// TIA Portal V20 export
TYPE "UDT_Tracability_Data"
   STRUCT
      Nb_of_Records { ExternalAccessible := 'False'; ExternalVisible := 'False'; ExternalWritable := 'False'} : Int := 100;
      Nb_of_Holes { ExternalAccessible := 'False'; ExternalVisible := 'False'; ExternalWritable := 'False'} : Int := 100;
      STRUCT_PART { ExternalAccessible := 'False'; ExternalVisible := 'False'; ExternalWritable := 'False'} : Array[0..99] of Struct
         Part_id : Int;
         Status : Int;
         Fail_code : Int;
         Raw_type : Int;
         Workpiece_holder_type : Int;
         Workpiece_holder_Nbr : Int;
         Datamatrix_code : Array[0..19] of Byte;
         Order_nbr : String[64];
         Ident_nbr : String[64];
         Batch_nbr : String[64];
         Operator_nbr : String[64];
         Comment : String[192];
         WOZ : Real;
         WOC : Real;
         Total_cycle_time : Int;
         Laser_cycle_time : Int;
         Measure_load_cycle_time : Int;
         STRUCT_HOLE : Array[0..99] of "UDT_Holes";
      END_STRUCT;
   END_STRUCT;
   // STRUCT_PART[1..10].Part_id := -1;
END_TYPE
